DATA_BLOCK "DATA"
VAR
  HaveAxisStart : Bool;
  AxisStartNumber : Int;
  "Forced modification" : Bool;
END_VAR
BEGIN
END_DATA_BLOCK
